# B&R Automation Studio project SW
Automation Studio 3.0.81.27 SP05

## Configuration Conveyor

CPU , AutomationRuntime M3.09, Build 4.1.2, Vc V4.05.4

### Task classes (Cpu.sw)
```
Cyclic#4 (cycle 100000 us, tolerance 100000 us):
  Stop_at_Li <- Stop_at_Lightsensor.prg
DataObjects: Acp10sys, arsdmhtm, arsdmsvg, arsdmsvp
Binaries: arsdm, ncglobal, Acp10man, webserv, acp10par, sysconf, ashwd, asfw, iomap, arconfig, Acp10map, Acp10cfg
Libraries: sys_lib, brsystem, Runtime, astcp, dataobj, powerlnk, astime, fileio, asmem, convert
```

### Hardware
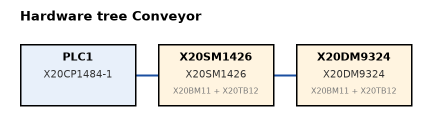
```
PLC1 : X20CP1484-1 v1.1.2.0
  Connector IF2:
    ActivateDevice = 1
  TimerDeviceType = EPLX2X
  TimerDevice = PLC1.IF6
  TaskClassIdleTime = 2000
  Cyclic1Duration = 2000
  Cyclic1Tolerance = 0
  Cyclic1Output = 1
  Cyclic2Duration = 20000
  Cyclic2Tolerance = 20000
  Cyclic3Duration = 50000
  Cyclic3Tolerance = 50000
  Cyclic4Duration = 100000
  Cyclic4Tolerance = 100000
  Cyclic5Duration = 200000
  Cyclic5Tolerance = 200000
  Cyclic6Duration = 500000
  Cyclic6Tolerance = 500000
  Cyclic7Duration = 1000000
  Cyclic7Tolerance = 1000000
  Cyclic8Duration = 10000
  Cyclic8Tolerance = 30000000
X20BM11 : X20BM11 v1.0.0.0  [X2X1 -> PLC1.IF6]
X20BM11a : X20BM11 v1.0.0.0  [X2X1 -> X20BM11.X2X2]
X20DM9324 : X20DM9324 v1.0.1.0  [SS1 -> X20TB12a.SS; SL -> X20BM11a.SL1]
  Supervision = off
  StatusInfo = off
X20SM1426 : X20SM1426 v1.3.2.0  [SS1 -> X20TB12.SS; SL -> X20BM11.SL1]
  FunctionModel = Ramp
  RatedCurrent01 = 70
  MaximumCurrent01 = 80
  MaxSpeed01pos_conf = 11250
  MaxAcc01_conf = 1280
  MaxDec01_conf = 1280
X20TB12 : X20TB12 v1.0.0.0
X20TB12a : X20TB12 v1.0.0.0
```

### IoMap.iom - PLC1/IoMap.iom
```iecst
(********************************************************************
 * COPYRIGHT --
 ********************************************************************
 * File: IoMap.iom
 * Author: Administrator
 * Created: October 24, 2011
 ********************************************************************
 * IO mapping file
 ********************************************************************)
VAR_CONFIG
	gaoControlword AT %QW."X20SM1426".MpGenControl01;
	gaiStatusword AT %IW."X20SM1426".MpGenStatus01;
	gaoMotorMode AT %QB."X20SM1426".MpGenMode01;
	gaiPos AT %ID."X20SM1426".AbsPos01ActVal;
	gaoVelocity AT %QD."X20SM1426".AbsPos01;
	gdiEmergencyOn AT %IX."X20DM9324".DigitalInput01;
	gdiOperating AT %IX."X20DM9324".DigitalInput02;
	gdiStart AT %IX."X20DM9324".DigitalInput03;
	gdiStop AT %IX."X20DM9324".DigitalInput04;
	gdiLightSensor1 AT %IX."X20DM9324".DigitalInput05;
	gdiLightSensor2 AT %IX."X20DM9324".DigitalInput06;
	gdiLightSensor3 AT %IX."X20DM9324".DigitalInput07;
	gdoStartLight AT %QX."X20DM9324".DigitalOutput01;
	gdoStopLight AT %QX."X20DM9324".DigitalOutput02;
	gdoPneumaticCylinder AT %QX."X20DM9324".DigitalOutput03;
END_VAR
```

## Configuration Conveyor_Simulation

CPU , AutomationRuntime D4.05, Build 4.1.2, Vc V4.05.4

### Task classes (Cpu.sw)
```
Cyclic#1 (cycle 100000 us, tolerance 10000000 us):
  Conveyor_S <- Conveyor_Simulator.prg
  Stop_at_Li <- Stop_at_Lightsensor.prg
DataObjects: arsdmhtm, arsdmsvg, arsdmsvp
Binaries: webserv, arsdm, sysconf, ashwd, arconfig, asfw
Libraries: runtime, astcp, dataobj, fileio, asmem, astime, convert, sys_lib
```

### Hardware
```
PLC1 : PC_any v1.1.0.0 (OrderNumber=PC)
  VolatileGlobalPvSize = 4096
  XLinkUseDefault = 0
  Cyclic1Duration = 100000
  Cyclic1Tolerance = 10000000
  Cyclic2Duration = 200000
  Cyclic2Tolerance = 10000000
  Cyclic3Duration = 500000
  Cyclic3Tolerance = 10000000
  Cyclic4Duration = 1000000
  Cyclic4Tolerance = 10000000
  Cyclic5Duration = 2000000
  Cyclic5Tolerance = 10000000
  Cyclic6Duration = 3000000
  Cyclic6Tolerance = 12000000
  Cyclic7Duration = 4000000
  Cyclic7Tolerance = 12000000
  Cyclic8Duration = 5000000
  Cyclic8Tolerance = 30000000
```

## Logical view

Binary libraries used (declarations not repeated): Convert, runtime, operator, sys_lib, brsystem, asstring

### Global.var - Global variables
```iecst
(********************************************************************
 * COPYRIGHT --
 ********************************************************************
 * File: Global.var
 * Author: Christoph Gruber
 * Created: October 24, 2011
 ********************************************************************
 * Global variables of project Foerderband
 ********************************************************************)
VAR
	gdiEmergencyOn : BOOL := FALSE;
	gdiOperating : BOOL := FALSE;
	gdiStart : BOOL := FALSE;
	gdoStartLight : BOOL := FALSE;
	gdiStop : BOOL := FALSE;
	gdoStopLight : BOOL := FALSE;
	gdiLightSensor3 : BOOL := FALSE;
	gdiLightSensor1 : BOOL := FALSE;
	gdiLightSensor2 : BOOL := FALSE;
	gdoPneumaticCylinder : BOOL := FALSE;
	gaoControlword : UINT := 0; (** ... see Help > Hardware > X20 System > X20 Modules > Motor modules > SM1426 > Register description of the ramp function model*)
	gaiStatusword : UINT := 0; (***)
	gaoMotorMode : SINT := 0; (***)
	gaoVelocity : DINT := 0; (*microsteps/MOTOR_MODULE_CYLCE_TIME*)
	gaiPos : DINT := 0; (*microsteps*)
END_VAR
```

### Global.h
```c
/********************************************************************
 * COPYRIGHT --
 ********************************************************************
 * Package: Conveyor
 * File: Global.h
 * Author: Christoph Gruber
 * Created: November 16, 2011
 *******************************************************************/

#include <bur/plctypes.h>
#define STATUS_READY_TO_SWITCH_ON          1
#define STATUS_SWITCHED_ON                 3
#define STATUS_OPERATION_ENABLED           7
#define CONTROL_SHUTDOWN                   6
#define CONTROL_SWITCH_ON                  7
#define CONTROL_OPERATION_ENABLE          15
#define MOTOR_VELOCITY_MODE                2
#define MOTOR_MODULE_CYCLE_TIME           25 /* ms */
#define SIMULATOR_TASK_CLASS_CYCLE_TIME  100 /* ms */
```


### Program Logical/Stop_at_Lightsensor (ANSIC) - Demo Program

#### Stop_at_LightsensorCyclic.c - Cyclic code
```c
/********************************************************************
 * COPYRIGHT --
 ********************************************************************
 * Program: Stop_at_Lightsensor
 * File: Stop_at_LightsensorCyclic.c
 * Author: Christoph Gruber
 * Created: October 24, 2011
 ********************************************************************
 * Implementation of program Stop_at_Lightsensor
 ********************************************************************/

#include <../Global.h>

#ifdef _DEFAULT_INCLUDES
 #include <AsDefault.h>
#endif

void _INIT Stop_at_LightsensorInit( void )
{
	gaoMotorMode = 2;
}

void _CYCLIC Stop_at_LightsensorCyclic( void )
{
	unsigned int motor_status = gaiStatusword & 0x0000000f;

	if (motor_status == STATUS_OPERATION_ENABLED)
	{
		if (!gdiLightSensor1)
		{
			gaoVelocity = 1000;
		}
		else
		{
			gaoVelocity = 0;
		}
	}
	else
	{
		switch (motor_status)
		{
		case STATUS_SWITCHED_ON:
			gaoControlword = CONTROL_OPERATION_ENABLE;
			break;
		case STATUS_READY_TO_SWITCH_ON:
			gaoControlword = CONTROL_SWITCH_ON;
			break;
		default:
			gaoControlword = CONTROL_SHUTDOWN;
		}
	}
}
```

### Program Logical/Conveyor_Simulator (ANSIC) - Simulator of the Conveyor Hardware

#### Conveyor_SimulatorCyclic.c - Cyclic code
```c
/********************************************************************
 * COPYRIGHT --
 ********************************************************************
 * Program: Conveyor_Simulator
 * File: Conveyor_SimulatorCyclic.c
 * Author: Christoph Gruber
 * Created: November 15, 2011
 ********************************************************************
 * Implementation of program Conveyor_Simulator
 ********************************************************************/

#include <../Global.h>

#ifdef _DEFAULT_INCLUDES
 #include <AsDefault.h>
#endif

void _INIT Conveyor_SimulatorInit( void )
{
	gaiPos = 0;
	gaiStatusword = STATUS_READY_TO_SWITCH_ON;
	gdiLightSensor1 = 0;
	gdiLightSensor2 = 0;
	gdiLightSensor3 = 0;
	gdiOperating = 0;
	gdiStart = 0;
	gdiStop = 0;
}

void _CYCLIC Conveyor_SimulatorCyclic( void )
{
	/* Motor Simulation */
	unsigned int controlword = old_controlword; /* Lets the motor module remain in the previous state for one more cycle*/
	old_controlword = gaoControlword;
	switch(controlword)
	{
	case CONTROL_SHUTDOWN:
		gaiStatusword = STATUS_READY_TO_SWITCH_ON;
		break;
	case CONTROL_SWITCH_ON:
		if (gaiStatusword == STATUS_READY_TO_SWITCH_ON)
			gaiStatusword = STATUS_SWITCHED_ON;
		break;
	case CONTROL_OPERATION_ENABLE:
		if (gaiStatusword == STATUS_SWITCHED_ON)
			gaiStatusword = STATUS_OPERATION_ENABLED;
		break;
	default:
		break;
	}

	if ((gaoMotorMode == MOTOR_VELOCITY_MODE) && (gaiStatusword == STATUS_OPERATION_ENABLED))
	{
		gaiPos = gaiPos + gaoVelocity / MOTOR_MODULE_CYCLE_TIME * SIMULATOR_TASK_CLASS_CYCLE_TIME;
	}
}
```

#### Conveyor_Simulator.var - Local variables
```iecst
(********************************************************************
 * COPYRIGHT --
 ********************************************************************
 * Program: Conveyor_Simulator
 * File: Conveyor_Simulator.var
 * Author: Christoph Gruber
 * Created: November 15, 2011
 ********************************************************************
 * Local variables of program Conveyor_Simulator
 ********************************************************************)
VAR
	old_controlword : UINT := 0;
END_VAR
```
